(* Logix 5000 project; controller lab6_LefeversAngelino 5069-L306ERM rev 30.11; software revision 30.00 *)

TASK MainTask (continuous, watchdog 500 ms) : MainProgram

MODULES
   Local : 5069-L306ERM (5069 0, rev 30.11)
      DudeBesideMe : 5069-L306ERM (Ethernet 10.14.1.15, rev 30.1, $c8a6b013$ RPI 20 ms)
      DudeBehindMe : 5069-L306ERM (Ethernet 10.14.1.5, rev 30.1, $e3c88687$ RPI 20 ms, $23548359$ RPI 20 ms)
      Analog_IN : vendor 1 type 115 code 314 (5069 2, rev 2.1, StandardDataDriven RPI 100 ms)
      Digital_IN : 5069-IB16 (5069 1, rev 2.1, StandardDataDriven RPI 5 ms)
      Analog_OUT : vendor 1 type 115 code 320 (5069 4, rev 2.1, StandardDataDriven RPI 80 ms)
      Digital_OUT : 5069-OB16 (5069 3, rev 2.1, StandardDataDriven RPI 5 ms)
END_MODULES

VAR_GLOBAL   (* controller tags *)
   BS : BOOL;
   LF1 : REAL[11] := ([10] := 1.0);
   LF2 : REAL[11] := ([10] := 1.0);
   MJ : REAL;   // PYT - Pretty Young Thing
   MOT1 : REAL := 966.1058;   // Motor Voltage Mine
   MOTOR_INPUT : REAL := 74.83696; {produced}   // Motor Volltage Other Guys
   MSG : MESSAGE;
        MessageParameters(ServiceCode := 16#004d, LocalElement := LF1[0], ...)
   MSG1 : MESSAGE;
        MessageParameters(ServiceCode := 16#004d, LocalElement := Local:2:I.Ch01.Data, ...)
   OJ : REAL := 244.10081;   // FREE OJ!!!!
   TEMP1 : REAL := 231.81738; {produced}   // Thermister Voltage Mine
   TEMP2 : REAL := 244.98918;   // Thermister Voltage His
   TEMP3 : REAL := 219.66887;   // Thermister Voltage Other Guy
   TM2 : TIMER := (PRE := 1000);
END_VAR

PROGRAM MainProgram   (* main routine MainRoutine *)
VAR
   CON1 : CONTROL := (LEN := 10, EM := 1);
   CON2 : CONTROL := (LEN := 10);
   GreenButton : ALIAS FOR Local:1:I.Pt01.Data;   // Normally Off
   Motor : ALIAS FOR Local:4:O.Ch01.Data;
   Potentiometer : ALIAS FOR Local:2:I.Ch00.Data;
   RedButton : ALIAS FOR Local:1:I.Pt00.Data;   // Normally On
   RedLED : ALIAS FOR Local:3:O.Pt00.Data;
   Thermister : ALIAS FOR Local:2:I.Ch01.Data;
   TM1 : TIMER := (PRE := 3000);
   TM3 : TIMER := (PRE := 1000, ACC := 8, EN := 1, TT := 1);
   ToggleLeft : ALIAS FOR Local:1:I.Pt03.Data;
   ToggleRight : ALIAS FOR Local:1:I.Pt02.Data;
END_VAR

ROUTINE MainRoutine   (* ladder *)
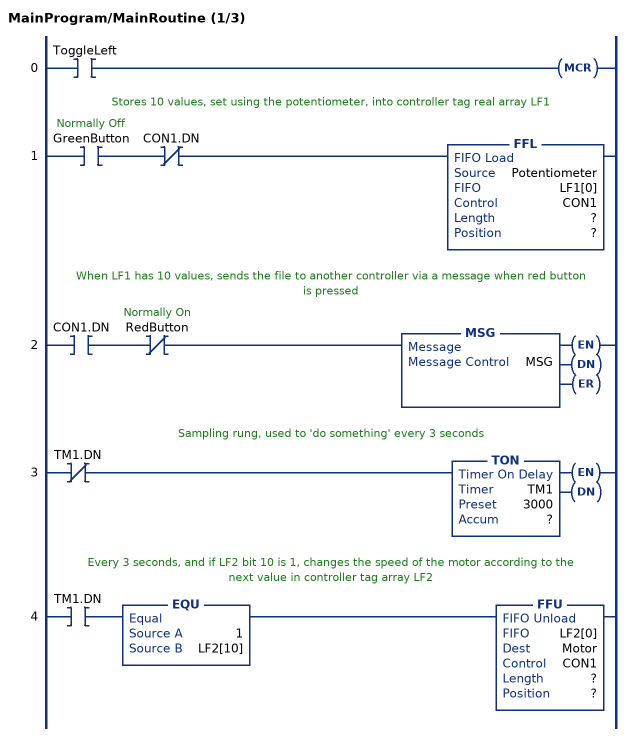
   0: XIC(ToggleLeft)MCR();
   // Stores 10 values, set using the potentiometer, into controller tag real array LF1
   1: XIC(GreenButton)XIO(CON1.DN)FFL(Potentiometer,LF1[0],CON1,?,?);
   // When LF1 has 10 values, sends the file to another controller via a message when red button is pressed
   2: XIC(CON1.DN)XIO(RedButton)MSG(MSG);
   // Sampling rung, used to 'do something' every 3 seconds
   3: XIO(TM1.DN)TON(TM1,?,?);
   // Every 3 seconds, and if LF2 bit 10 is 1, changes the speed of the motor according to the next value in controller tag array LF2
   4: XIC(TM1.DN)EQU(1,LF2[10])FFU(LF2[0],Motor,CON1,?,?);
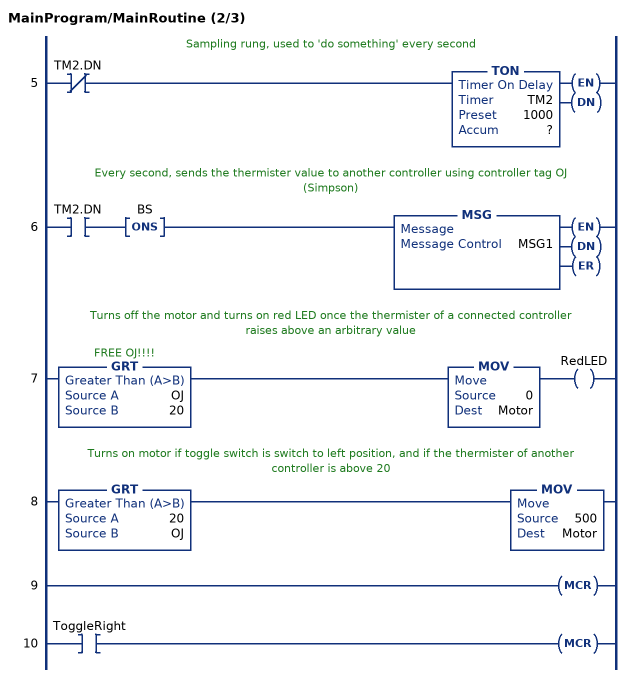
   // Sampling rung, used to 'do something' every second
   5: XIO(TM2.DN)TON(TM2,?,?);
   // Every second, sends the thermister value to another controller using controller tag OJ (Simpson)
   6: XIC(TM2.DN)ONS(BS)MSG(MSG1);
   // Turns off the motor and turns on red LED once the thermister of a connected controller raises above an arbitrary value
   7: GRT(OJ,20)MOV(0,Motor)OTE(RedLED);
   // Turns on motor if toggle switch is switch to left position, and if the thermister of another controller is above 20
   8: GRT(20,OJ)MOV(500,Motor);
   9: MCR();
   10: XIC(ToggleRight)MCR();
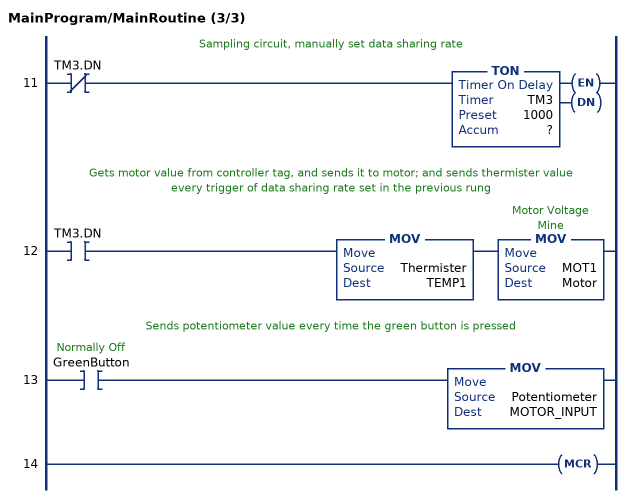
   // Sampling circuit, manually set data sharing rate
   11: XIO(TM3.DN)TON(TM3,?,?);
   // Gets motor value from controller tag, and sends it to motor; and sends thermister value every trigger of data sharing rate set in the previous rung
   12: XIC(TM3.DN)MOV(Thermister,TEMP1)MOV(MOT1,Motor);
   // Sends potentiometer value every time the green button is pressed
   13: XIC(GreenButton)MOV(Potentiometer,MOTOR_INPUT);
   14: MCR();
END_ROUTINE
END_PROGRAM
